// SIMATIC S7-200 project (STEP 7-Micro/WIN), CPU 224 CN REL 02.01

ORGANIZATION_BLOCK 主程序:OB1
TITLE=程序注释
BEGIN
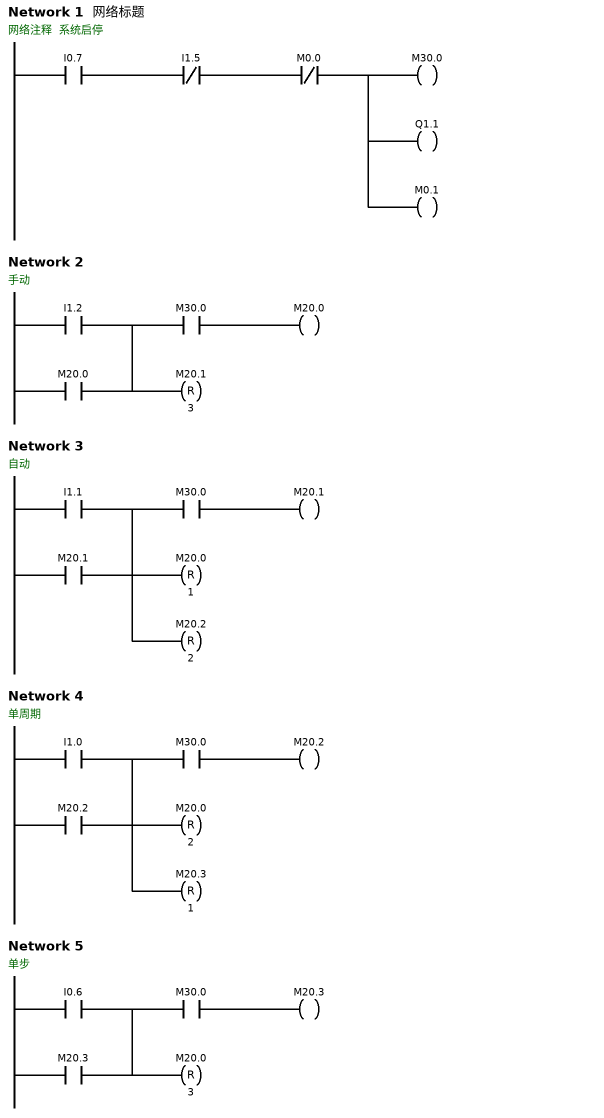
Network 1 // 网络标题
// 网络注释	系统启停
LD     I0.7
AN     I1.5
AN     M0.0
=      M30.0
=      Q1.1
=      M0.1
Network 2
// 手动	
LD     I1.2
O      M20.0
LPS
A      M30.0
=      M20.0
LPP
R      M20.1, 3
Network 3
// 自动
LD     I1.1
O      M20.1
LPS
A      M30.0
=      M20.1
LRD
R      M20.0, 1
LPP
R      M20.2, 2
Network 4
// 单周期
LD     I1.0
O      M20.2
LPS
A      M30.0
=      M20.2
LRD
R      M20.0, 2
LPP
R      M20.3, 1
Network 5
// 单步
LD     I0.6
O      M20.3
LPS
A      M30.0
=      M20.3
LPP
R      M20.0, 3
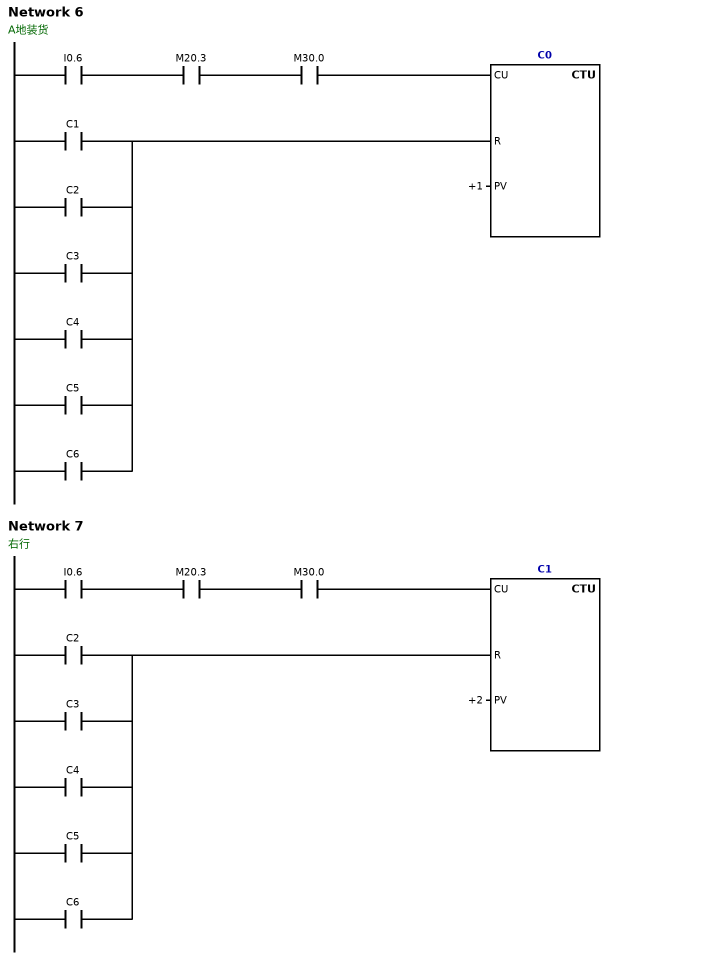
Network 6
// A地装货
LD     I0.6
A      M20.3
A      M30.0
LD     C1
O      C2
O      C3
O      C4
O      C5
O      C6
CTU    C0, +1
Network 7
// 右行
LD     I0.6
A      M20.3
A      M30.0
LD     C2
O      C3
O      C4
O      C5
O      C6
CTU    C1, +2
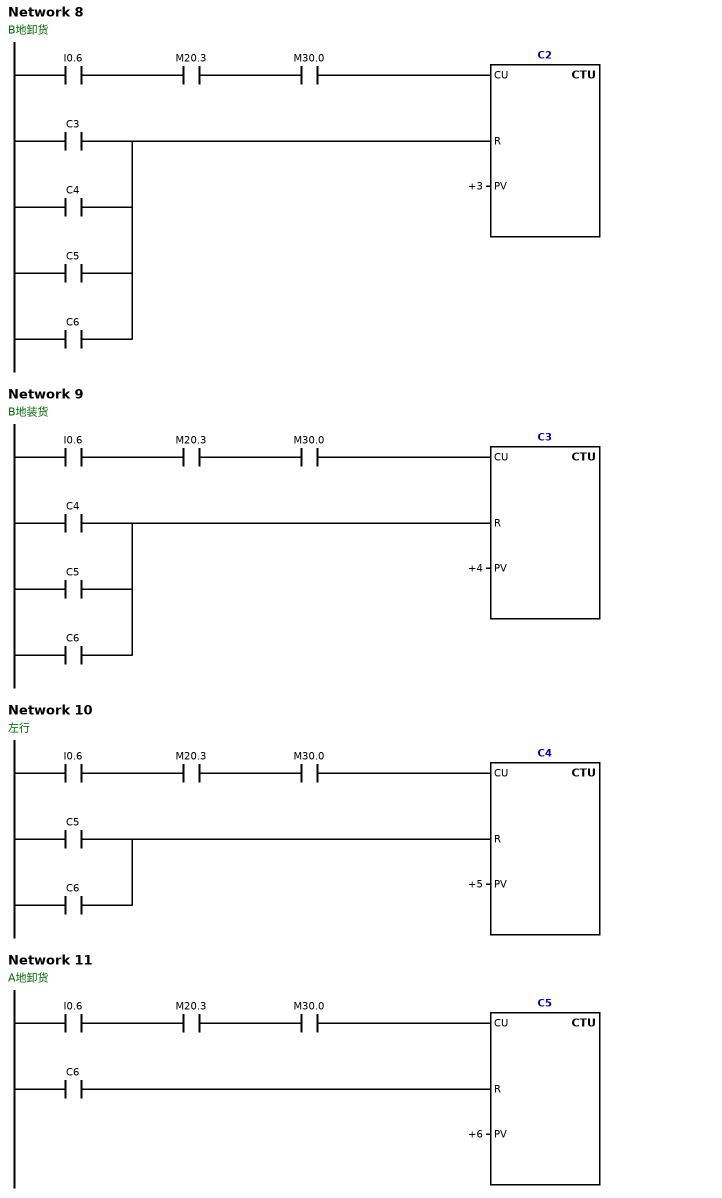
Network 8
// B地卸货
LD     I0.6
A      M20.3
A      M30.0
LD     C3
O      C4
O      C5
O      C6
CTU    C2, +3
Network 9
// B地装货
LD     I0.6
A      M20.3
A      M30.0
LD     C4
O      C5
O      C6
CTU    C3, +4
Network 10
// 左行
LD     I0.6
A      M20.3
A      M30.0
LD     C5
O      C6
CTU    C4, +5
Network 11
// A地卸货
LD     I0.6
A      M20.3
A      M30.0
LD     C6
CTU    C5, +6
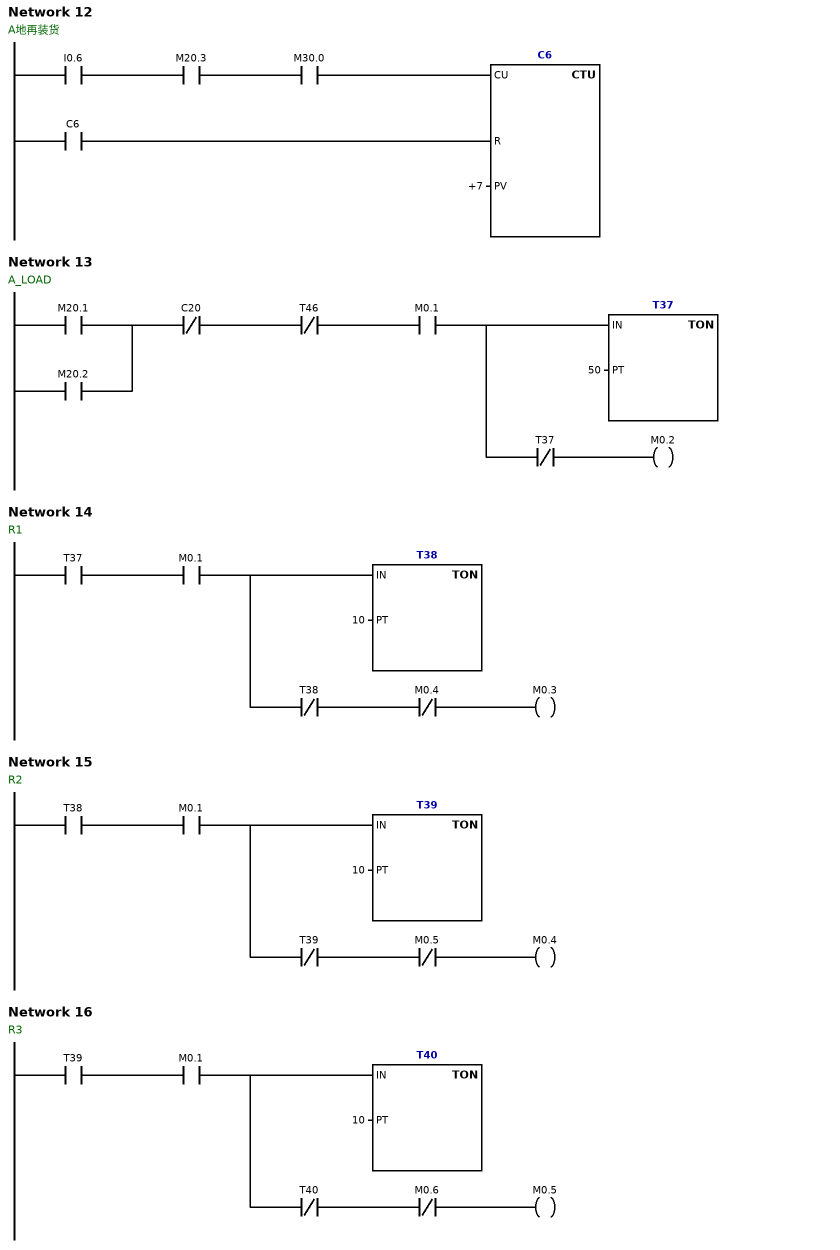
Network 12
// A地再装货
LD     I0.6
A      M20.3
A      M30.0
LD     C6
CTU    C6, +7
Network 13
// A_LOAD
LD     M20.1
O      M20.2
AN     C20
AN     T46
A      M0.1
TON    T37, 50
AN     T37
=      M0.2
Network 14
// R1
LD     T37
A      M0.1
TON    T38, 10
AN     T38
AN     M0.4
=      M0.3
Network 15
// R2
LD     T38
A      M0.1
TON    T39, 10
AN     T39
AN     M0.5
=      M0.4
Network 16
// R3
LD     T39
A      M0.1
TON    T40, 10
AN     T40
AN     M0.6
=      M0.5
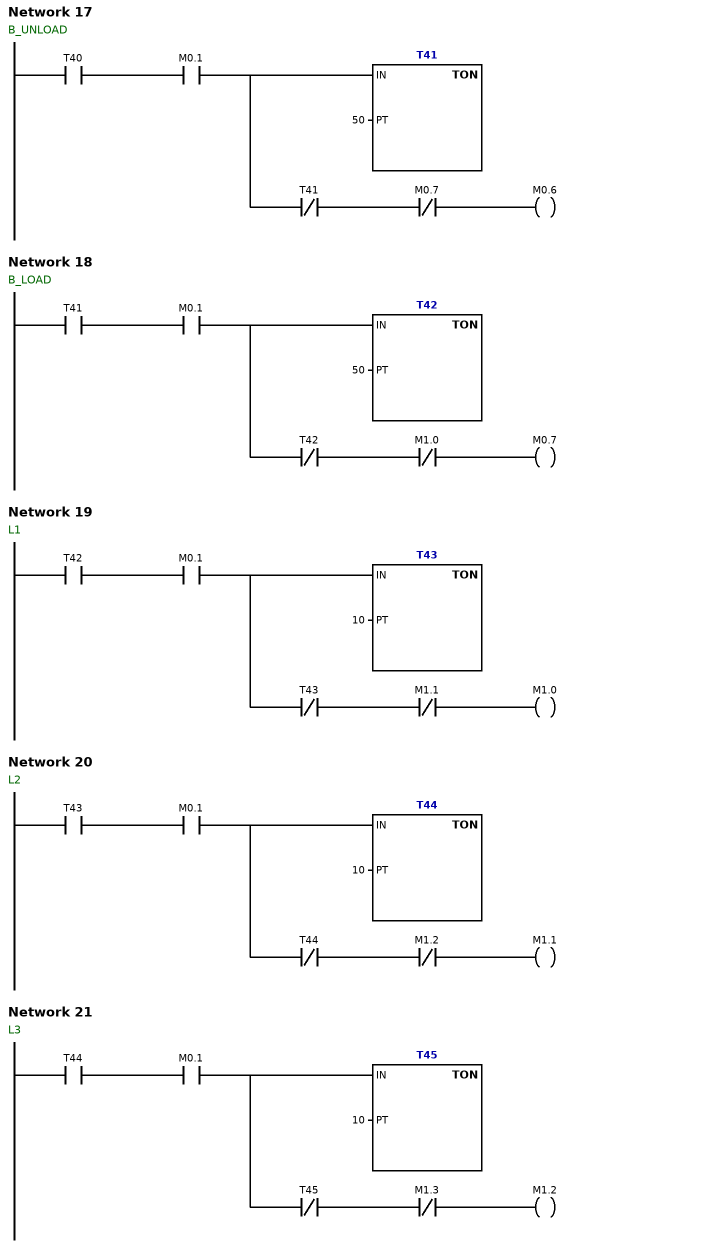
Network 17
// B_UNLOAD
LD     T40
A      M0.1
TON    T41, 50
AN     T41
AN     M0.7
=      M0.6
Network 18
// B_LOAD
LD     T41
A      M0.1
TON    T42, 50
AN     T42
AN     M1.0
=      M0.7
Network 19
// L1
LD     T42
A      M0.1
TON    T43, 10
AN     T43
AN     M1.1
=      M1.0
Network 20
// L2
LD     T43
A      M0.1
TON    T44, 10
AN     T44
AN     M1.2
=      M1.1
Network 21
// L3
LD     T44
A      M0.1
TON    T45, 10
AN     T45
AN     M1.3
=      M1.2
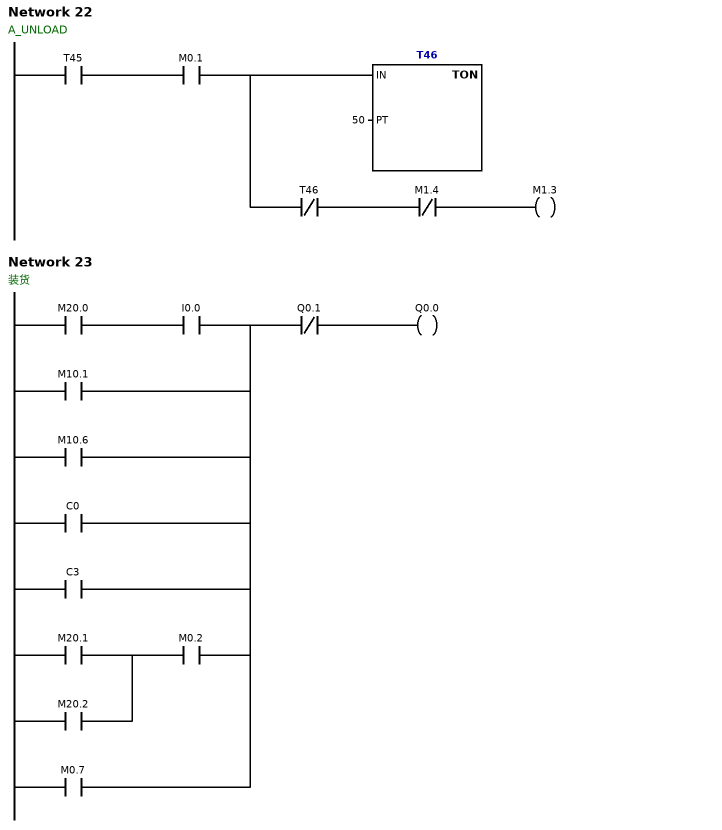
Network 22
// A_UNLOAD
LD     T45
A      M0.1
TON    T46, 50
AN     T46
AN     M1.4
=      M1.3
Network 23
// 装货
LD     M20.0
A      I0.0
O      M10.1
O      M10.6
O      C0
O      C3
LD     M20.1
O      M20.2
A      M0.2
OLD
O      M0.7
AN     Q0.1
=      Q0.0
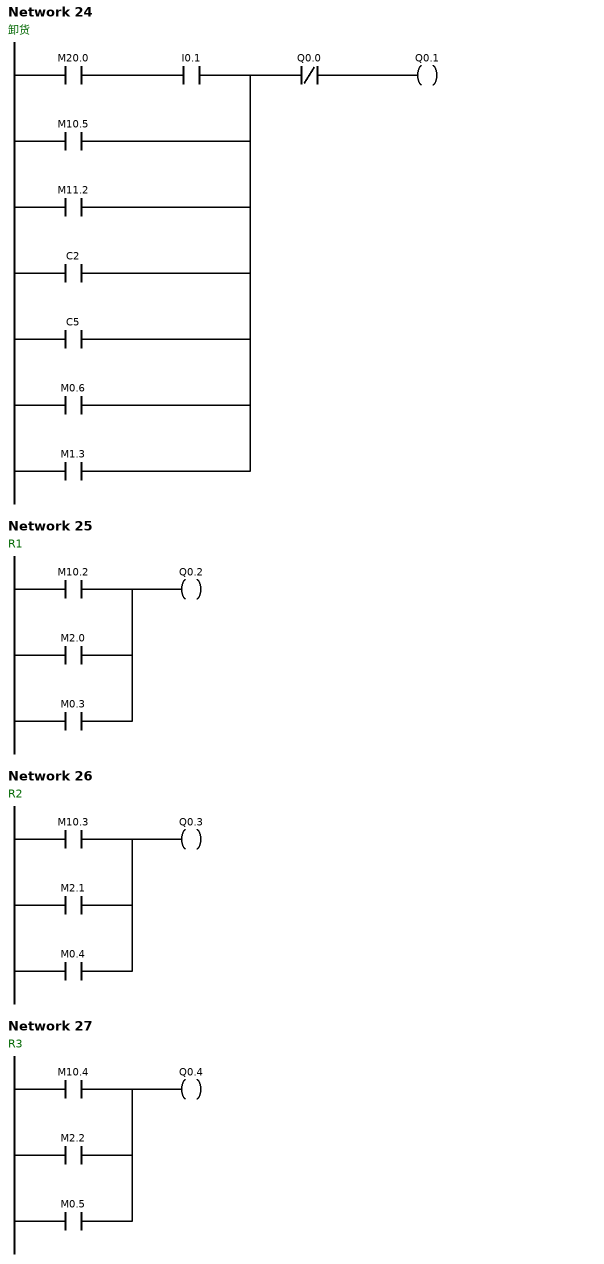
Network 24
// 卸货
LD     M20.0
A      I0.1
O      M10.5
O      M11.2
O      C2
O      C5
O      M0.6
O      M1.3
AN     Q0.0
=      Q0.1
Network 25
// R1
LD     M10.2
O      M2.0
O      M0.3
=      Q0.2
Network 26
// R2
LD     M10.3
O      M2.1
O      M0.4
=      Q0.3
Network 27
// R3
LD     M10.4
O      M2.2
O      M0.5
=      Q0.4
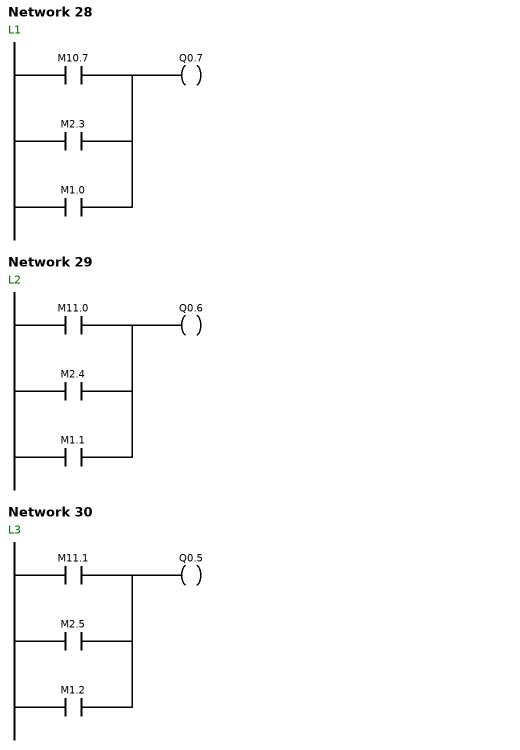
Network 28
// L1
LD     M10.7
O      M2.3
O      M1.0
=      Q0.7
Network 29
// L2
LD     M11.0
O      M2.4
O      M1.1
=      Q0.6
Network 30
// L3
LD     M11.1
O      M2.5
O      M1.2
=      Q0.5
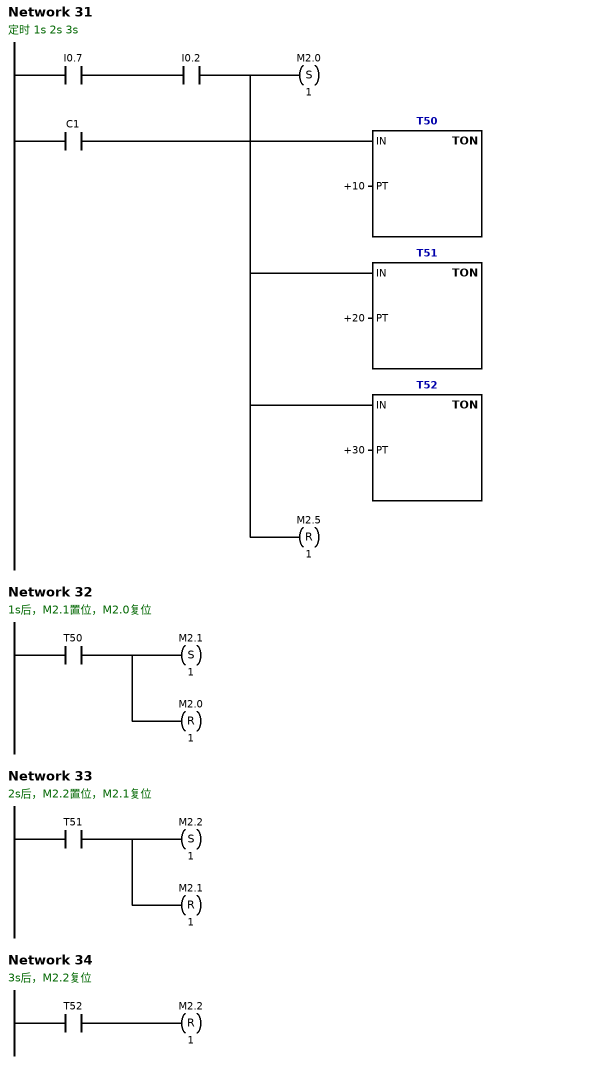
Network 31
// 定时 1s 2s 3s
LD     I0.7
A      I0.2
O      C1
S      M2.0, 1
TON    T50, +10
TON    T51, +20
TON    T52, +30
R      M2.5, 1
Network 32
// 1s后，M2.1置位，M2.0复位
LD     T50
S      M2.1, 1
R      M2.0, 1
Network 33
// 2s后，M2.2置位，M2.1复位
LD     T51
S      M2.2, 1
R      M2.1, 1
Network 34
// 3s后，M2.2复位
LD     T52
R      M2.2, 1
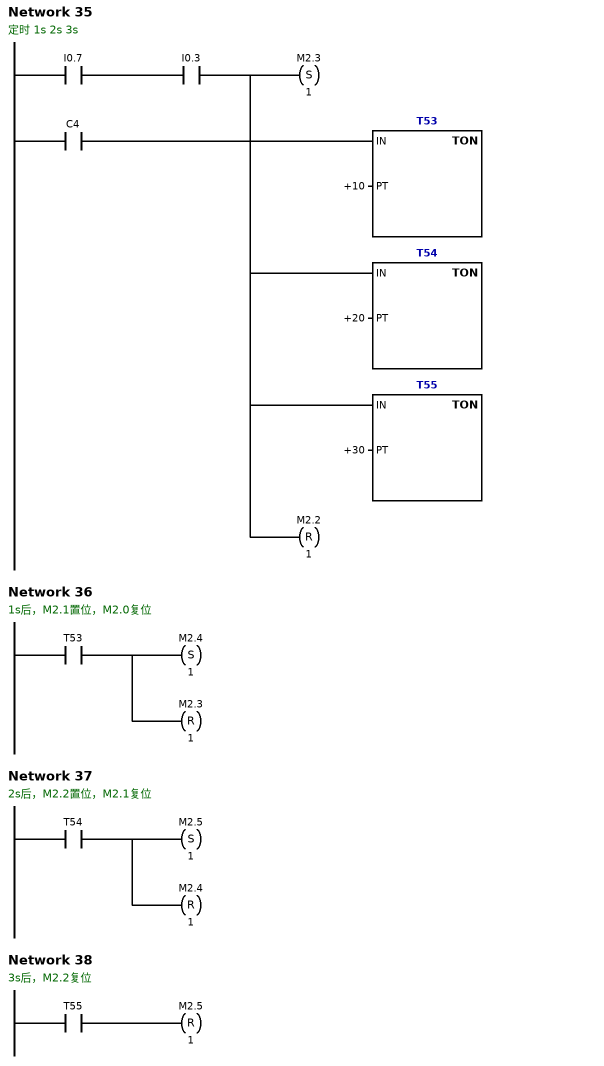
Network 35
// 定时 1s 2s 3s
LD     I0.7
A      I0.3
O      C4
S      M2.3, 1
TON    T53, +10
TON    T54, +20
TON    T55, +30
R      M2.2, 1
Network 36
// 1s后，M2.1置位，M2.0复位
LD     T53
S      M2.4, 1
R      M2.3, 1
Network 37
// 2s后，M2.2置位，M2.1复位
LD     T54
S      M2.5, 1
R      M2.4, 1
Network 38
// 3s后，M2.2复位
LD     T55
R      M2.5, 1
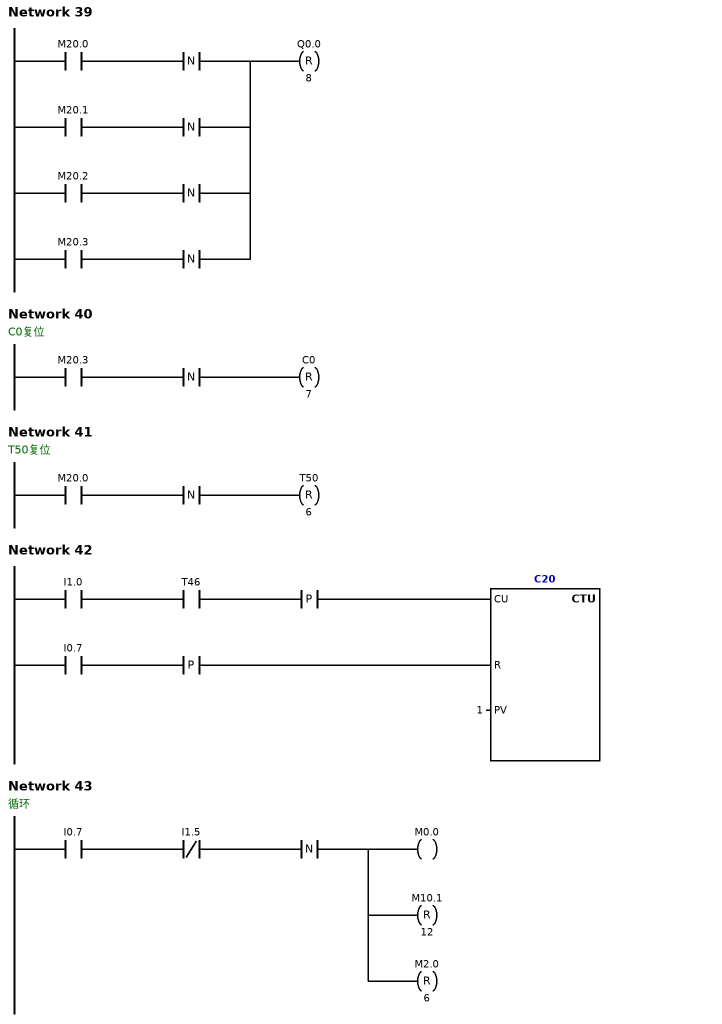
Network 39
LD     M20.0
ED
LD     M20.1
ED
OLD
LD     M20.2
ED
OLD
LD     M20.3
ED
OLD
R      Q0.0, 8
Network 40
// C0复位
LD     M20.3
ED
R      C0, 7
Network 41
// T50复位
LD     M20.0
ED
R      T50, 6
Network 42
LD     I1.0
A      T46
EU
LD     I0.7
EU
CTU    C20, 1
Network 43
// 循环
LD     I0.7
AN     I1.5
ED
=      M0.0
R      M10.1, 12
R      M2.0, 6
END_ORGANIZATION_BLOCK
